{attribute 'qualified_only'}
{attribute 'strict'}
TYPE MC_StartMode :
(
	mcAbsolute := 0,
	mcRelative := 1,
	mcRampIn := 2
);
END_TYPE

(* stored: Version 1.1.0.1, ProductVersion 3.1.4024.12
   DUT MC_StartMode: Id {b8737406-d6b2-458b-876f-182ae35279a3} *)
